(* IEC 61131-3 sources: AXOpen/src/components.festo.drives/ctrl/src/AxoCmmtAs (part 7) *)

            IF(_AxisReference = NULL) THEN
                RETURN;
            END_IF;

            IF Enable THEN
                Busy := TRUE;
                IF VelocityFactor <= 0.0 OR  VelocityFactor >= 2.0 OR AccelerationFactor <= 0.0 OR  AccelerationFactor > 1.0 OR JerkFactor <= 0.0 OR  JerkFactor > 1.0 THEN
                    Error := TRUE;
                ELSE
                    _AxisReference^.Data.OverrideVelocityFactor := VelocityFactor;
                    _AxisReference^.Data.OverrideAccelerationFactor := AccelerationFactor;
                    _AxisReference^.Data.OverrideJerkFactor := JerkFactor;
                    _AxisReference^.Telegram111_Out.Override_ := TO_WORD(TO_INT(16384.0/VelocityFactor));
                    Enabled	:= TRUE;
                END_IF;
            END_IF;
        END_METHOD

        ///<summary>
        /// This method returns the value of a vendor specific parameter. The returned Value has to be converted to Real
        /// if necessary. If not possible, the vendor has to supply a vendor specific method to read the parameter.
        ///<summary>
        VAR INTERNAL
            MC_ReadParameterEnable_PV       : 	BOOL := FALSE;		//Enable - previous value
            MC_ReadParameterErrorID         : 	WORD;
            MC_ReadParameterCycle			: 	ULINT;
            MC_ReadParameterValue			: 	LINT;
            MC_ReadParameterValid			: 	BOOL;
        END_VAR
        METHOD PUBLIC OVERRIDE MC_ReadParameter
            VAR_INPUT
                AxisRef         :   AXOpen.Components.Abstractions.Drives.IAxoAxisReference;
                Enable          :   BOOL;                       //  Get the value of the parameter continuously while enabled
                ParameterNumber :   DINT;                       //  Number of the parameter. One can also use symbolic parameter names which are declared as VAR CONST.
            END_VAR
            VAR_OUTPUT
                Valid           :   BOOL;                       //  A valid output is available at the method
                Busy            :   BOOL;                       //  The method is not finished and new output values are to be expected
                Error           :   BOOL;                       //  Signals that an error has occurred within the method
                ErrorID         :   WORD;                       //  Error identification
                Value           :   LINT;                       //  Value of the specified parameter in the datatype, as specified by the vendor
            END_VAR
            VAR
                _AxisReference :  REF_TO AXOpen.Components.Festo.Drives.AxoCmmtAsAxisReference;
                Dummy : BOOL;
            END_VAR

            _AxisReference ?= AxisRef;

            Messenger.ActivateOnCondition(ULINT#720,_AxisReference = NULL, eAxoMessageCategory#ProgrammingError);

            IF(_AxisReference = NULL) THEN
                RETURN;
            END_IF;

            IF Enable AND NOT MC_ReadParameterEnable_PV AND State = UINT#0 THEN
                _AxisReference^.Status.CurrentMotionTaskId := AXOpen.Components.Drives.eAxoMotionTaskId#Axo_ReadParameter;
                _AxisReference^.Data.Cycle := _AxisReference^.Data.Cycle + ULINT#2;
                MC_ReadParameterCycle := _AxisReference^.Data.Cycle ;
            END_IF;

            IF Enable THEN
                IF State = UINT#0 THEN
                    Busy := TRUE;
                    MC_ReadParameterErrorID := WORD#16#0000;
                    Parametrization.Inputs.Enable := FALSE;
                    State := UINT#160;
                END_IF;
                IF State = UINT#160 THEN
                    Busy := TRUE;
                    Parametrization.Inputs.Enable := TRUE;
                    Parametrization.Inputs.ReadWrite   := FALSE;
                    Parametrization.Inputs.ParameterNo := TO_INT(ParameterNumber);
                    Parametrization.Inputs.Subindex    := 0;
                    Parametrization.Inputs.AxisNo  := BYTE#1;
                    Parametrization.Inputs.HardwareId  := _AxisReference^.Data.MAP_HW_ID;
                    IF Parametrization.Outputs.Done AND NOT Parametrization.Outputs.Error THEN
                        MC_ReadParameterValid := TRUE;
                        MC_ReadParameterValue := Parametrization.Outputs.ValueReadLINT;
                        State := UINT#161;
                    END_IF;
                    IF Parametrization.Outputs.Error THEN
                        MC_MoveVelocityErrorID := WORD#801;
                        State := UINT#169;
                    END_IF;
                END_IF;
                IF State = UINT#161 THEN
                    Busy := TRUE;
                    Parametrization.Inputs.Enable := FALSE;
                    Parametrization.Inputs.ReadWrite   := FALSE;
                    IF  NOT Parametrization.Outputs.Done THEN
                        State := UINT#160;
                    END_IF;
                END_IF;
                IF State = UINT#169 THEN
                    Error := TRUE;
                END_IF;

                IF State>=UINT#160 AND State<UINT#167 THEN
                    IF _AxisReference^.Data.Cycle <> MC_ReadParameterCycle THEN
                        _AxisReference^.Data.Cycle := _AxisReference^.Data.Cycle - ULINT#1;
                        State := UINT#169;
                    END_IF;
                END_IF;
            END_IF;

            IF NOT Enable AND MC_ReadParameterEnable_PV  THEN
                _AxisReference^.Status.CurrentMotionTaskId := AXOpen.Components.Drives.eAxoMotionTaskId#Axo_None;
                MC_ReadParameterErrorID := WORD#0;
                MC_ReadParameterCycle := ULINT#0;
                MC_ReadParameterValid := FALSE;
                MC_ReadParameterValue := LINT#0;
                State := UINT#0;
            END_IF;

            ErrorID := MC_ReadParameterErrorID;
            Valid := MC_ReadParameterValid;
            Value := MC_ReadParameterValue;
            MC_ReadParameterEnable_PV := Enable;
        END_METHOD

        ///<summary>
        /// This method returns the value of a vendor specific parameter with datatype REAL.
        ///<summary>
        VAR INTERNAL
            MC_ReadRealParameterEnable_PV       : 	BOOL := FALSE;		//Enable - previous value
            MC_ReadRealParameterErrorID         : 	WORD;
            MC_ReadRealParameterCycle			: 	ULINT;
            MC_ReadRealParameterValue			: 	REAL;
            MC_ReadRealParameterValid			: 	BOOL;
        END_VAR
        METHOD PUBLIC OVERRIDE MC_ReadRealParameter
            VAR_INPUT
                AxisRef         :   AXOpen.Components.Abstractions.Drives.IAxoAxisReference;
                Enable          :   BOOL;                       //  Get the value of the parameter continuously while enabled
                ParameterNumber :   DINT;                       //  Number of the parameter. One can also use symbolic parameter names which are declared as VAR CONST.
            END_VAR
            VAR_OUTPUT
                Valid           :   BOOL;                       //  A valid output is available at the method
                Busy            :   BOOL;                       //  The method is not finished and new output values are to be expected
                Error           :   BOOL;                       //  Signals that an error has occurred within the method
                ErrorID         :   WORD;                       //  Error identification
                Value           :   REAL;                       //  Value of the specified parameter in the datatype, as specified by the vendor
            END_VAR
            VAR
                _AxisReference :  REF_TO AXOpen.Components.Festo.Drives.AxoCmmtAsAxisReference;
                Dummy : BOOL;
            END_VAR

            _AxisReference ?= AxisRef;

            Messenger.ActivateOnCondition(ULINT#721,_AxisReference = NULL, eAxoMessageCategory#ProgrammingError);

            IF(_AxisReference = NULL) THEN
                RETURN;
            END_IF;
            IF Enable AND NOT MC_ReadRealParameterEnable_PV AND State = UINT#0 THEN
                _AxisReference^.Status.CurrentMotionTaskId := AXOpen.Components.Drives.eAxoMotionTaskId#Axo_ReadRealParameter;
                _AxisReference^.Data.Cycle := _AxisReference^.Data.Cycle + ULINT#2;
                MC_ReadRealParameterCycle := _AxisReference^.Data.Cycle ;
            END_IF;

            IF Enable THEN
                IF State = UINT#0 THEN
                    Busy := TRUE;
                    MC_ReadRealParameterErrorID := WORD#16#0000;
                    Parametrization.Inputs.Enable := FALSE;
                    State := UINT#170;
                END_IF;
                IF State = UINT#170 THEN
                    Busy := TRUE;
                    Parametrization.Inputs.Enable := TRUE;
                    Parametrization.Inputs.ReadWrite   := FALSE;
                    Parametrization.Inputs.ParameterNo := TO_INT(ParameterNumber);
                    Parametrization.Inputs.Subindex    := 0;
                    Parametrization.Inputs.AxisNo  := BYTE#1;
                    Parametrization.Inputs.HardwareId  := _AxisReference^.Data.MAP_HW_ID;
                    IF Parametrization.Outputs.Done AND NOT Parametrization.Outputs.Error THEN
                        MC_ReadRealParameterValid := TRUE;
                        MC_ReadRealParameterValue := Parametrization.Outputs.ValueReadREAL;
                        State := UINT#171;
                    END_IF;
                    IF Parametrization.Outputs.Error THEN
                        MC_MoveVelocityErrorID := WORD#802;
                        State := UINT#179;
                    END_IF;
                END_IF;
                IF State = UINT#171 THEN
                    Busy := TRUE;
                    Parametrization.Inputs.Enable := FALSE;
                    Parametrization.Inputs.ReadWrite   := FALSE;
                    IF  NOT Parametrization.Outputs.Done THEN
                        State := UINT#170;
                    END_IF;
                END_IF;
                IF State = UINT#179 THEN
                    Error := TRUE;
                END_IF;

                IF State>=UINT#170 AND State<UINT#177 THEN
                    IF _AxisReference^.Data.Cycle <> MC_ReadRealParameterCycle THEN
                        _AxisReference^.Data.Cycle := _AxisReference^.Data.Cycle - ULINT#1;
                        State := UINT#179;
                    END_IF;
                END_IF;
            END_IF;

            IF NOT Enable AND MC_ReadRealParameterEnable_PV  THEN
                _AxisReference^.Status.CurrentMotionTaskId := AXOpen.Components.Drives.eAxoMotionTaskId#Axo_None;
                MC_ReadRealParameterErrorID := WORD#0;
                MC_ReadRealParameterCycle := ULINT#0;
                MC_ReadRealParameterValid := FALSE;
                MC_ReadRealParameterValue := REAL#0.0;
                State := UINT#0;
            END_IF;

            ErrorID := MC_ReadRealParameterErrorID;
            Valid := MC_ReadRealParameterValid;
            Value := MC_ReadRealParameterValue;
            MC_ReadRealParameterEnable_PV := Enable;
        END_METHOD

        ///<summary>
        /// This method returns the value of a vendor specific parameter with datatype BOOL.
        ///<summary>
        VAR INTERNAL
            MC_ReadBoolParameterEnable_PV       : 	BOOL := FALSE;		//Enable - previous value
            MC_ReadBoolParameterErrorID         : 	WORD;
            MC_ReadBoolParameterCycle			: 	ULINT;
            MC_ReadBoolParameterValue			: 	BOOL;
            MC_ReadBoolParameterValid			: 	BOOL;
        END_VAR
        METHOD PUBLIC OVERRIDE MC_ReadBoolParameter
            VAR_INPUT
                AxisRef         :   AXOpen.Components.Abstractions.Drives.IAxoAxisReference;
                Enable          :   BOOL;                       //  Get the value of the parameter continuously while enabled
                ParameterNumber :   DINT;                       //  Number of the parameter. One can also use symbolic parameter names which are declared as VAR CONST.
            END_VAR
            VAR_OUTPUT
                Valid           :   BOOL;                       //  A valid output is available at the method
                Busy            :   BOOL;                       //  The method is not finished and new output values are to be expected
                Error           :   BOOL;                       //  Signals that an error has occurred within the method
                ErrorID         :   WORD;                       //  Error identification
                Value           :   BOOL;                       //  Value of the specified parameter in the datatype, as specified by the vendor
            END_VAR
            VAR
                _AxisReference :  REF_TO AXOpen.Components.Festo.Drives.AxoCmmtAsAxisReference;
                Dummy : BOOL;
            END_VAR
            RETURN;

            _AxisReference ?= AxisRef;

            Messenger.ActivateOnCondition(ULINT#722,_AxisReference = NULL, eAxoMessageCategory#ProgrammingError);

            IF(_AxisReference = NULL) THEN
                RETURN;
            END_IF;

            IF Enable AND NOT MC_ReadBoolParameterEnable_PV AND State = UINT#0 THEN
                _AxisReference^.Status.CurrentMotionTaskId := AXOpen.Components.Drives.eAxoMotionTaskId#Axo_ReadBoolParameter;
                _AxisReference^.Data.Cycle := _AxisReference^.Data.Cycle + ULINT#2;
                MC_ReadBoolParameterCycle := _AxisReference^.Data.Cycle ;
            END_IF;

            IF Enable THEN
                IF State = UINT#0 THEN
                    Busy := TRUE;
                    MC_ReadBoolParameterErrorID := WORD#16#0000;
                    Parametrization.Inputs.Enable := FALSE;
                    State := UINT#180;
                END_IF;
                IF State = UINT#180 THEN
                    Busy := TRUE;
                    Parametrization.Inputs.Enable := TRUE;
                    Parametrization.Inputs.ReadWrite   := FALSE;
                    Parametrization.Inputs.ParameterNo := TO_INT(ParameterNumber);
                    Parametrization.Inputs.Subindex    := 0;
                    Parametrization.Inputs.AxisNo  := BYTE#1;
                    Parametrization.Inputs.HardwareId  := _AxisReference^.Data.MAP_HW_ID;
                    IF Parametrization.Outputs.Done AND NOT Parametrization.Outputs.Error THEN
                        MC_ReadBoolParameterValid := TRUE;
                        MC_ReadBoolParameterValue := Parametrization.Outputs.ValueReadBOOL;
                        State := UINT#181;
                    END_IF;
                    IF Parametrization.Outputs.Error THEN
                        MC_MoveVelocityErrorID := WORD#801;
                        State := UINT#189;
                    END_IF;
                END_IF;
                IF State = UINT#181 THEN
                    Busy := TRUE;
                    Parametrization.Inputs.Enable := FALSE;
                    Parametrization.Inputs.ReadWrite   := FALSE;
                    IF  NOT Parametrization.Outputs.Done THEN
                        State := UINT#180;
                    END_IF;
                END_IF;
                IF State = UINT#189 THEN
                    Error := TRUE;
                END_IF;

                IF State>=UINT#180 AND State<UINT#187 THEN
                    IF _AxisReference^.Data.Cycle <> MC_ReadBoolParameterCycle THEN
                        _AxisReference^.Data.Cycle := _AxisReference^.Data.Cycle - ULINT#1;
                        State := UINT#189;
                    END_IF;
                END_IF;
            END_IF;

            IF NOT Enable AND MC_ReadBoolParameterEnable_PV  THEN
                _AxisReference^.Status.CurrentMotionTaskId := AXOpen.Components.Drives.eAxoMotionTaskId#Axo_None;
                MC_ReadBoolParameterErrorID := WORD#0;
                MC_ReadBoolParameterCycle := ULINT#0;
                MC_ReadBoolParameterValid := FALSE;
                MC_ReadBoolParameterValue := FALSE;
                State := UINT#0;
            END_IF;

            ErrorID := MC_ReadBoolParameterErrorID;
            Valid := MC_ReadBoolParameterValid;
            Value := MC_ReadBoolParameterValue;
            MC_ReadBoolParameterEnable_PV := Enable;

        END_METHOD

        ///<summary>
        /// This method modifies the value of a vendor specific parameter.
        ///<summary>
        VAR INTERNAL
            MC_WriteParameterExecute_PV     : 	BOOL := FALSE;		//Enable - previous value
            MC_WriteParameterErrorID        : 	WORD;
            MC_WriteParameterCycle			: 	ULINT;
        END_VAR
        METHOD PUBLIC OVERRIDE MC_WriteParameter
            VAR_INPUT
                AxisRef         :   AXOpen.Components.Abstractions.Drives.IAxoAxisReference;
                Execute         :   BOOL;                       //  Write the value of the parameter at rising edge
                ParameterNumber :   DINT;                       //  Number of the parameter (correspondence between number andparameter is specified in the table above)
                Value           :   LINT;                       //  New value of the specified parameter
                ExecutionMode   :   AXOpen.Components.Abstractions.Drives.eAxoExecutionMode;          //  Defines the chronological sequence of the method.
            END_VAR
            VAR_OUTPUT
                Done            :   BOOL;                       //  Parameter successfully written
                Busy            :   BOOL;                       //  The method is not finished and new output values are to be expected.
                Error           :   BOOL;                       //  Signals that an error has occurred within the method
                ErrorID         :   WORD;                       //  Error identification
            END_VAR
            VAR
                _AxisReference :  REF_TO AXOpen.Components.Festo.Drives.AxoCmmtAsAxisReference;
                Dummy : BOOL;
            END_VAR

            _AxisReference ?= AxisRef;

            Messenger.ActivateOnCondition(ULINT#723,_AxisReference = NULL, eAxoMessageCategory#ProgrammingError);

            IF(_AxisReference = NULL) THEN
                RETURN;
            END_IF;

            IF THIS.AxoWriteParameter_Task.StartTriggered()  THEN
                _AxisReference^.Status.CurrentMotionTaskId := AXOpen.Components.Drives.eAxoMotionTaskId#Axo_WriteParameter;
            END_IF;

            IF Execute AND NOT MC_WriteParameterExecute_PV AND State = UINT#0 THEN
                _AxisReference^.Data.Cycle := _AxisReference^.Data.Cycle + ULINT#2;
                MC_WriteParameterCycle := _AxisReference^.Data.Cycle ;
            END_IF;

            IF Execute THEN
                IF State = UINT#0 THEN
                    Busy := TRUE;
                    Parametrization.Inputs.Enable := FALSE;
                    State := UINT#190;
                END_IF;
                IF State = UINT#190 THEN
                    Busy := TRUE;
                    Parametrization.Inputs.Enable := TRUE;
                    Parametrization.Inputs.ReadWrite   := TRUE;
                    Parametrization.Inputs.ParameterNo := TO_INT(ParameterNumber);
                    Parametrization.Inputs.Subindex    := 0;
                    Parametrization.Inputs.AxisNo  := BYTE#1;
                    Parametrization.Inputs.HardwareId  := _AxisReference^.Data.MAP_HW_ID;
                    Parametrization.Inputs.ValueWriteLINT := Value;
                    IF Parametrization.Outputs.Done AND NOT Parametrization.Outputs.Error THEN
                        State := UINT#191;
                    END_IF;
                    IF Parametrization.Outputs.Error THEN
                        MC_WriteParameterErrorID := WORD#804;
                        State := UINT#199;
                    END_IF;
                END_IF;
                IF State = UINT#191 THEN
                    Busy := TRUE;
                    Parametrization.Inputs.Enable := FALSE;
                    Parametrization.Inputs.ReadWrite   := FALSE;
                    IF  NOT Parametrization.Outputs.Done THEN
                        State := UINT#197;
                    END_IF;
                END_IF;
                IF State = UINT#197 THEN
                    Done := TRUE;
                    MC_WriteParameterCycle := ULINT#0;
                END_IF;
                IF State = UINT#199 THEN
                    MC_WriteParameterCycle := ULINT#0;
                    Error := TRUE;
                END_IF;

                IF State>=UINT#190 AND State<UINT#197 THEN
                    IF _AxisReference^.Data.Cycle <> MC_WriteParameterCycle THEN
                        _AxisReference^.Data.Cycle := _AxisReference^.Data.Cycle - ULINT#1;
                        State := UINT#199;
                    END_IF;
                END_IF;
            END_IF;

            IF THIS.AxoWriteParameter_Task.DoneReached() THEN
                _AxisReference^.Status.CurrentMotionTaskId := AXOpen.Components.Drives.eAxoMotionTaskId#Axo_Done;
                MC_WriteParameterErrorID := WORD#0;
                // MC_WriteParameterCycle := ULINT#0;
                State := UINT#0;
            END_IF;

            IF THIS.AxoWriteParameter_Task.RestoreTriggered() AND State>=UINT#190 AND State<=UINT#199 THEN
                _AxisReference^.Status.CurrentMotionTaskId := AXOpen.Components.Drives.eAxoMotionTaskId#Axo_None;
                MC_WriteParameterErrorID := WORD#0;
                MC_WriteParameterCycle := ULINT#0;
                State := UINT#0;
            END_IF;

            ErrorID := MC_WriteParameterErrorID;
            MC_WriteParameterExecute_PV := Execute;
        END_METHOD

        ///<summary>
        /// This method modifies the value of a vendor specific parameter of type Real.
        ///<summary>
        VAR INTERNAL
            MC_WriteRealParameterExecute_PV     : 	BOOL := FALSE;		//Enable - previous value
            MC_WriteRealParameterErrorID        : 	WORD;
            MC_WriteRealParameterCycle			: 	ULINT;
        END_VAR
        METHOD PUBLIC OVERRIDE MC_WriteRealParameter
            VAR_INPUT
                AxisRef         :   AXOpen.Components.Abstractions.Drives.IAxoAxisReference;
                Execute         :   BOOL;                       //  Write the value of the parameter at rising edge
                ParameterNumber :   DINT;                       //  Number of the parameter (correspondence between number andparameter is specified in the table above)
                Value           :   REAL;                       //  New value of the specified parameter
                ExecutionMode   :   AXOpen.Components.Abstractions.Drives.eAxoExecutionMode;          //  Defines the chronological sequence of the method.
            END_VAR
            VAR_OUTPUT
                Done            :   BOOL;                       //  Parameter successfully written
                Busy            :   BOOL;                       //  The method is not finished and new output values are to be expected.
                Error           :   BOOL;                       //  Signals that an error has occurred within the method
                ErrorID         :   WORD;                       //  Error identification
            END_VAR
            VAR
                _AxisReference :  REF_TO AXOpen.Components.Festo.Drives.AxoCmmtAsAxisReference;
                Dummy : BOOL;
            END_VAR

            _AxisReference ?= AxisRef;

            Messenger.ActivateOnCondition(ULINT#724,_AxisReference = NULL, eAxoMessageCategory#ProgrammingError);

            IF(_AxisReference = NULL) THEN
                RETURN;
            END_IF;

            IF THIS.AxoWriteRealParameter_Task.StartTriggered()  THEN
                _AxisReference^.Status.CurrentMotionTaskId := AXOpen.Components.Drives.eAxoMotionTaskId#Axo_WriteRealParameter;
            END_IF;

            IF Execute AND NOT MC_WriteRealParameterExecute_PV AND State = UINT#0 THEN
                _AxisReference^.Data.Cycle := _AxisReference^.Data.Cycle + ULINT#2;
                MC_WriteRealParameterCycle := _AxisReference^.Data.Cycle ;
            END_IF;

            IF Execute THEN
                IF State = UINT#0 THEN
                    Busy := TRUE;
                    Parametrization.Inputs.Enable := FALSE;
                    State := UINT#200;
                END_IF;
                IF State = UINT#200 THEN
                    Busy := TRUE;
                    Parametrization.Inputs.Enable := TRUE;
                    Parametrization.Inputs.ReadWrite   := TRUE;
                    Parametrization.Inputs.ParameterNo := TO_INT(ParameterNumber);
                    Parametrization.Inputs.Subindex    := 0;
                    Parametrization.Inputs.AxisNo  := BYTE#1;
                    Parametrization.Inputs.HardwareId  := _AxisReference^.Data.MAP_HW_ID;
                    Parametrization.Inputs.ValueWriteREAL := Value;
                    IF Parametrization.Outputs.Done AND NOT Parametrization.Outputs.Error THEN
                        State := UINT#201;
                    END_IF;
                    IF Parametrization.Outputs.Error THEN
                        MC_WriteRealParameterErrorID := WORD#805;
                        State := UINT#209;
                    END_IF;
                END_IF;
                IF State = UINT#201 THEN
                    Busy := TRUE;
                    Parametrization.Inputs.Enable := FALSE;
                    Parametrization.Inputs.ReadWrite   := FALSE;
                    IF  NOT Parametrization.Outputs.Done THEN
                        State := UINT#207;
                    END_IF;
                END_IF;
                IF State = UINT#207 THEN
                    Done := TRUE;
                    MC_WriteRealParameterCycle := ULINT#0;
                END_IF;
                IF State = UINT#209 THEN
                    MC_WriteRealParameterCycle := ULINT#0;
                    Error := TRUE;
                END_IF;

                IF State>=UINT#200 AND State<UINT#207 THEN
                    IF _AxisReference^.Data.Cycle <> MC_WriteRealParameterCycle THEN
                        _AxisReference^.Data.Cycle := _AxisReference^.Data.Cycle - ULINT#1;
                        State := UINT#209;
                    END_IF;
                END_IF;
            END_IF;

            IF THIS.AxoWriteRealParameter_Task.DoneReached() THEN
                _AxisReference^.Status.CurrentMotionTaskId := AXOpen.Components.Drives.eAxoMotionTaskId#Axo_Done;
                MC_WriteRealParameterErrorID := WORD#0;
                // MC_WriteRealParameterCycle := ULINT#0;
                State := UINT#0;
            END_IF;

            IF THIS.AxoWriteRealParameter_Task.RestoreTriggered() AND State>=UINT#200 AND State<=UINT#209 THEN
                _AxisReference^.Status.CurrentMotionTaskId := AXOpen.Components.Drives.eAxoMotionTaskId#Axo_None;
                MC_WriteRealParameterErrorID := WORD#0;
                MC_WriteRealParameterCycle := ULINT#0;
                State := UINT#0;
            END_IF;

            ErrorID := MC_WriteRealParameterErrorID;
            MC_WriteRealParameterExecute_PV := Execute;
        END_METHOD

        ///<summary>
        /// This method modifies the value of a vendor specific parameter of type BOOL.
        ///<summary>
        VAR INTERNAL
            MC_WriteBoolParameterExecute_PV     : 	BOOL := FALSE;		//Enable - previous value
            MC_WriteBoolParameterErrorID        : 	WORD;
            MC_WriteBoolParameterCycle			: 	ULINT;
        END_VAR
        METHOD PUBLIC OVERRIDE MC_WriteBoolParameter
            VAR_INPUT
                AxisRef         :   AXOpen.Components.Abstractions.Drives.IAxoAxisReference;
                Execute         :   BOOL;                       //  Write the value of the parameter at rising edge
                ParameterNumber :   DINT;                       //  Number of the parameter (correspondence between number andparameter is specified in the table above)
                Value           :   BOOL;                       //  New value of the specified parameter
                ExecutionMode   :   AXOpen.Components.Abstractions.Drives.eAxoExecutionMode;          //  Defines the chronological sequence of the method.
            END_VAR
            VAR_OUTPUT
                Done            :   BOOL;                       //  Parameter successfully written
                Busy            :   BOOL;                       //  The method is not finished and new output values are to be expected.
                Error           :   BOOL;                       //  Signals that an error has occurred within the method
                ErrorID         :   WORD;                       //  Error identification
            END_VAR
            VAR
                _AxisReference :  REF_TO AXOpen.Components.Festo.Drives.AxoCmmtAsAxisReference;
                Dummy : BOOL;
            END_VAR

            _AxisReference ?= AxisRef;

            Messenger.ActivateOnCondition(ULINT#725,_AxisReference = NULL, eAxoMessageCategory#ProgrammingError);

            IF(_AxisReference = NULL) THEN
                RETURN;
            END_IF;

            IF THIS.AxoWriteBoolParameter_Task.StartTriggered()  THEN
                _AxisReference^.Status.CurrentMotionTaskId := AXOpen.Components.Drives.eAxoMotionTaskId#Axo_WriteBoolParameter;
            END_IF;

            IF Execute AND NOT MC_WriteBoolParameterExecute_PV AND State = UINT#0 THEN
                _AxisReference^.Data.Cycle := _AxisReference^.Data.Cycle + ULINT#2;
                MC_WriteBoolParameterCycle := _AxisReference^.Data.Cycle ;
            END_IF;

            IF Execute THEN
                IF State = UINT#0 THEN
                    Busy := TRUE;
                    Parametrization.Inputs.Enable := FALSE;
                    State := UINT#210;
                END_IF;
                IF State = UINT#210 THEN
                    Busy := TRUE;
                    Parametrization.Inputs.Enable := TRUE;
                    Parametrization.Inputs.ReadWrite   := TRUE;
                    Parametrization.Inputs.ParameterNo := TO_INT(ParameterNumber);
                    Parametrization.Inputs.Subindex    := 0;
                    Parametrization.Inputs.AxisNo  := BYTE#1;
                    Parametrization.Inputs.HardwareId  := _AxisReference^.Data.MAP_HW_ID;
                    Parametrization.Inputs.ValueWriteBOOL := Value;
                    IF Parametrization.Outputs.Done AND NOT Parametrization.Outputs.Error THEN
                        State := UINT#211;
                    END_IF;
                    IF Parametrization.Outputs.Error THEN
                        MC_WriteBoolParameterErrorID := WORD#805;
                        State := UINT#219;
                    END_IF;
                END_IF;
                IF State = UINT#211 THEN
                    Busy := TRUE;
                    Parametrization.Inputs.Enable := FALSE;
                    Parametrization.Inputs.ReadWrite   := FALSE;
                    IF  NOT Parametrization.Outputs.Done THEN
                        State := UINT#217;
                    END_IF;
                END_IF;
                IF State = UINT#217 THEN
                    Done := TRUE;
                    MC_WriteBoolParameterCycle := ULINT#0;
                END_IF;
                IF State = UINT#219 THEN
                    MC_WriteBoolParameterCycle := ULINT#0;
                    Error := TRUE;
                END_IF;

                IF State>=UINT#210 AND State<UINT#217 THEN
                    IF _AxisReference^.Data.Cycle <> MC_WriteBoolParameterCycle THEN
                        _AxisReference^.Data.Cycle := _AxisReference^.Data.Cycle - ULINT#1;
                        State := UINT#219;
                    END_IF;
                END_IF;
            END_IF;

            IF THIS.AxoWriteBoolParameter_Task.DoneReached() THEN
                _AxisReference^.Status.CurrentMotionTaskId := AXOpen.Components.Drives.eAxoMotionTaskId#Axo_Done;
                MC_WriteBoolParameterErrorID := WORD#0;
                // MC_WriteBoolParameterCycle := ULINT#0;
                State := UINT#0;
            END_IF;

            IF THIS.AxoWriteBoolParameter_Task.RestoreTriggered() AND State>=UINT#210 AND State<=UINT#219 THEN
                _AxisReference^.Status.CurrentMotionTaskId := AXOpen.Components.Drives.eAxoMotionTaskId#Axo_None;
                MC_WriteBoolParameterErrorID := WORD#0;
                MC_WriteBoolParameterCycle := ULINT#0;
                State := UINT#0;
            END_IF;

            ErrorID := MC_WriteBoolParameterErrorID;
            MC_WriteBoolParameterExecute_PV := Execute;
        END_METHOD

        ///<summary>
        /// This method gives access to the value of the input, referenced by the datatype MC_INPUT_REF.
        /// It provides the value of the referenced input (BOOL).
        ///<summary>
        VAR INTERNAL
            MC_ReadDigitalInputEnable_PV        : 	BOOL := FALSE;		//Enable - previous value
            MC_ReadDigitalInputErrorID          : 	WORD;
            MC_ReadDigitalInputCycle			: 	ULINT;
            MC_ReadDigitalInputValue			: 	BOOL;
            MC_ReadDigitalInputValid			: 	BOOL;
        END_VAR
        METHOD PUBLIC OVERRIDE MC_ReadDigitalInput
            VAR_INPUT
                AxisRef         :   AXOpen.Components.Abstractions.Drives.IAxoAxisReference;
                Enable          :   BOOL;                       //  Get the value of the selected input signal continuously while enabled
                InputNumber     :   INT;                        //  Selects the input. Can be part of MC_INPUT_REF, if only one single input is referenced.
            END_VAR
            VAR_OUTPUT
                Valid           :   BOOL;                       //  A valid output is available at the method
                Busy            :   BOOL;                       //  The method is not finished and new output values are to be expected
                Error           :   BOOL;                       //  Signals that an error has occurred within the method
                ErrorID         :   WORD;                       //  Error identification
                Value           :   BOOL;                       //  The value of the selected input signal
            END_VAR
            VAR
                _AxisReference :  REF_TO AXOpen.Components.Festo.Drives.AxoCmmtAsAxisReference;
                Dummy : BOOL;
            END_VAR

            _AxisReference ?= AxisRef;

            Messenger.ActivateOnCondition(ULINT#726,_AxisReference = NULL, eAxoMessageCategory#ProgrammingError);

            IF(_AxisReference = NULL) THEN
                RETURN;
            END_IF;

            IF Enable AND NOT MC_ReadDigitalInputEnable_PV AND State = UINT#0 THEN
                _AxisReference^.Status.CurrentMotionTaskId := AXOpen.Components.Drives.eAxoMotionTaskId#Axo_ReadDigitalInput;
                _AxisReference^.Data.Cycle := _AxisReference^.Data.Cycle + ULINT#2;
                MC_ReadDigitalInputCycle := _AxisReference^.Data.Cycle ;
            END_IF;

            IF Enable THEN
                IF State = UINT#0 THEN
                    Busy := TRUE;
                    MC_ReadDigitalInputErrorID := WORD#16#0000;
                    Parametrization.Inputs.Enable := FALSE;
                    State := UINT#220;
                END_IF;
                IF State = UINT#220 THEN
                    Busy := TRUE;
                    Parametrization.Inputs.Enable := TRUE;
                    Parametrization.Inputs.ReadWrite   := FALSE;
                    Parametrization.Inputs.ParameterNo := 2888;
                    Parametrization.Inputs.Subindex    := 0;
                    Parametrization.Inputs.AxisNo  := BYTE#1;
                    Parametrization.Inputs.HardwareId  := _AxisReference^.Data.MAP_HW_ID;
                    IF Parametrization.Outputs.Done AND NOT Parametrization.Outputs.Error THEN
                        MC_ReadDigitalInputValid := TRUE;
                        MC_ReadDigitalInputValue := GetBit(TO_LWORD(Parametrization.Outputs.ValueReadLINT), TO_USINT(InputNumber));
                        State := UINT#221;
                    END_IF;
                    IF Parametrization.Outputs.Error THEN
                        MC_MoveVelocityErrorID := WORD#807;
                        State := UINT#229;
                    END_IF;
                END_IF;
                IF State = UINT#221 THEN
                    Busy := TRUE;
                    Parametrization.Inputs.Enable := FALSE;
                    Parametrization.Inputs.ReadWrite   := FALSE;
                    IF  NOT Parametrization.Outputs.Done THEN
                        State := UINT#220;
                    END_IF;
                END_IF;
                IF State = UINT#229 THEN
                    Error := TRUE;
                END_IF;

                IF State>=UINT#220 AND State<UINT#227 THEN
                    IF _AxisReference^.Data.Cycle <> MC_ReadDigitalInputCycle THEN
                        _AxisReference^.Data.Cycle := _AxisReference^.Data.Cycle - ULINT#1;
                        State := UINT#229;
                    END_IF;
                END_IF;
            END_IF;

            IF NOT Enable AND MC_ReadDigitalInputEnable_PV  THEN
                _AxisReference^.Status.CurrentMotionTaskId := AXOpen.Components.Drives.eAxoMotionTaskId#Axo_None;
                MC_ReadDigitalInputErrorID := WORD#0;
                MC_ReadDigitalInputCycle := ULINT#0;
                MC_ReadDigitalInputValid := FALSE;
                MC_ReadDigitalInputValue := FALSE;
                State := UINT#0;
            END_IF;

            ErrorID := MC_ReadDigitalInputErrorID;
            Valid := MC_ReadDigitalInputValid;
            Value := MC_ReadDigitalInputValue;
            MC_ReadDigitalInputEnable_PV := Enable;
        END_METHOD

        ///<summary>
        /// This method provides access to the value of a digital output, referenced by the datatype MC_OUTPUT_REF.
        /// It provides the value of the referenced output (BOOL).
        ///<summary>
        VAR INTERNAL
            MC_ReadDigitalOutputEnable_PV        : 	BOOL := FALSE;		//Enable - previous value
            MC_ReadDigitalOutputErrorID          : 	WORD;
            MC_ReadDigitalOutputCycle			: 	ULINT;
            MC_ReadDigitalOutputValue			: 	BOOL;
            MC_ReadDigitalOutputValid			: 	BOOL;
        END_VAR
        METHOD PUBLIC OVERRIDE MC_ReadDigitalOutput
            VAR_INPUT
                AxisRef         :   AXOpen.Components.Abstractions.Drives.IAxoAxisReference;
                Enable          :   BOOL;                       //  Get the value of the selected output signal continuously while enabled
                OutputNumber    :   INT;                        //  Selects the output. Can be part of MC_OUTPUT_REF, if only one single output is referenced.
            END_VAR
            VAR_OUTPUT
                Valid           :   BOOL;                       //  A valid output is available at the method
                Busy            :   BOOL;                       //  The method is not finished and new output values are to be expected
                Error           :   BOOL;                       //  Signals that an error has occurred within the method
                ErrorID         :   WORD;                       //  Error identification
                Value           :   BOOL;                       //  The value of the selected output signal
            END_VAR
            VAR
                _AxisReference :  REF_TO AXOpen.Components.Festo.Drives.AxoCmmtAsAxisReference;
                Dummy : BOOL;
            END_VAR

            _AxisReference ?= AxisRef;

            Messenger.ActivateOnCondition(ULINT#727,_AxisReference = NULL, eAxoMessageCategory#ProgrammingError);

            IF(_AxisReference = NULL) THEN
                RETURN;
            END_IF;

            IF Enable AND NOT MC_ReadDigitalOutputEnable_PV AND State = UINT#0 THEN
                _AxisReference^.Status.CurrentMotionTaskId := AXOpen.Components.Drives.eAxoMotionTaskId#Axo_ReadDigitalOutput;
                _AxisReference^.Data.Cycle := _AxisReference^.Data.Cycle + ULINT#2;
                MC_ReadDigitalOutputCycle := _AxisReference^.Data.Cycle ;
            END_IF;

            IF Enable THEN
                IF State = UINT#0 THEN
                    Busy := TRUE;
                    MC_ReadDigitalOutputErrorID := WORD#16#0000;
                    Parametrization.Inputs.Enable := FALSE;
                    State := UINT#230;
                END_IF;
                IF State = UINT#230 THEN
                    Busy := TRUE;
                    Parametrization.Inputs.Enable := TRUE;
                    Parametrization.Inputs.ReadWrite   := FALSE;
                    Parametrization.Inputs.ParameterNo := 2888;
                    Parametrization.Inputs.Subindex    := 0;
                    Parametrization.Inputs.AxisNo  := BYTE#1;
                    Parametrization.Inputs.HardwareId  := _AxisReference^.Data.MAP_HW_ID;
                    IF Parametrization.Outputs.Done AND NOT Parametrization.Outputs.Error THEN
                        MC_ReadDigitalOutputValid := TRUE;
                        MC_ReadDigitalOutputValue := GetBit(TO_LWORD(Parametrization.Outputs.ValueReadLINT), TO_USINT(OutputNumber));
                        State := UINT#231;
                    END_IF;
                    IF Parametrization.Outputs.Error THEN
                        MC_MoveVelocityErrorID := WORD#809;
                        State := UINT#239;
                    END_IF;
                END_IF;
                IF State = UINT#231 THEN
                    Busy := TRUE;
                    Parametrization.Inputs.Enable := FALSE;
                    Parametrization.Inputs.ReadWrite   := FALSE;
                    IF  NOT Parametrization.Outputs.Done THEN
                        State := UINT#230;
                    END_IF;
                END_IF;
                IF State = UINT#239 THEN
                    Error := TRUE;
                END_IF;

                IF State>=UINT#230 AND State<UINT#237 THEN
                    IF _AxisReference^.Data.Cycle <> MC_ReadDigitalOutputCycle THEN
                        _AxisReference^.Data.Cycle := _AxisReference^.Data.Cycle - ULINT#1;
                        State := UINT#239;
                    END_IF;
                END_IF;
            END_IF;

            IF NOT Enable AND MC_ReadDigitalOutputEnable_PV  THEN
                _AxisReference^.Status.CurrentMotionTaskId := AXOpen.Components.Drives.eAxoMotionTaskId#Axo_None;
                MC_ReadDigitalOutputErrorID := WORD#0;
                MC_ReadDigitalOutputCycle := ULINT#0;
                MC_ReadDigitalOutputValid := FALSE;
                MC_ReadDigitalOutputValue := FALSE;
                State := UINT#0;
            END_IF;

            ErrorID := MC_ReadDigitalOutputErrorID;
            Valid := MC_ReadDigitalOutputValid;
            Value := MC_ReadDigitalOutputValue;
            MC_ReadDigitalOutputEnable_PV := Enable;
        END_METHOD

        ///<summary>
        /// This method writes a value to the output referenced by the argument ‘Output’ once (with rising edge of Execute)
        ///<summary>
        VAR INTERNAL
            MC_WriteDigitalOutputExecute_PV     : 	BOOL := FALSE;		//Enable - previous value
            MC_WriteDigitalOutputErrorID        : 	WORD;
            MC_WriteDigitalOutputCycle			: 	ULINT;
        END_VAR
        METHOD PUBLIC OVERRIDE MC_WriteDigitalOutput
            VAR_INPUT
                AxisRef         :   AXOpen.Components.Abstractions.Drives.IAxoAxisReference;
                Execute         :   BOOL;                       //  Write the value of the selected output
                OutputNumber    :   INT;                        //  Selects the output. Can be part of MC_OUTPUT_REF, if only one single output is referenced.
                Value           :   BOOL;                       //  The value of the selected output signal
                ExecutionMode   :   AXOpen.Components.Abstractions.Drives.eAxoExecutionMode;          //  Defines the chronological sequence of the method.
            END_VAR
            VAR_OUTPUT
                Done            :   BOOL;                       //  Writing of the output signal value is done
                Busy            :   BOOL;                       //  The method is not finished and new output values are to be expected.
                Error           :   BOOL;                       //  Signals that an error has occurred within the method
                ErrorID         :   WORD;                       //  Error identification
            END_VAR
            VAR
                _AxisReference :  REF_TO AXOpen.Components.Festo.Drives.AxoCmmtAsAxisReference;
                Dummy : BOOL;
                Valid_          :   BOOL;
                Error_          :   BOOL;
                ErrorID_        :   WORD;
            END_VAR

            _AxisReference ?= AxisRef;

            Messenger.ActivateOnCondition(ULINT#728,_AxisReference = NULL, eAxoMessageCategory#ProgrammingError);

            IF(_AxisReference = NULL) THEN
                RETURN;
            END_IF;

            IF THIS.AxoWriteDigitalOutput_Task.StartTriggered()  THEN
                _AxisReference^.Status.CurrentMotionTaskId := AXOpen.Components.Drives.eAxoMotionTaskId#Axo_WriteDigitalOutput;
            END_IF;

            IF Execute AND NOT MC_WriteDigitalOutputExecute_PV AND State = UINT#0 THEN
                _AxisReference^.Data.Cycle := _AxisReference^.Data.Cycle + ULINT#2;
                MC_WriteDigitalOutputCycle := _AxisReference^.Data.Cycle ;
            END_IF;

            IF Execute THEN
                IF State = UINT#0 THEN
                    Busy := TRUE;
                    Parametrization.Inputs.Enable := FALSE;
                    State := UINT#240;
                    //Remove after implementation on the drive side
                    State := UINT#249;
                    MC_WriteDigitalOutputErrorID := WORD#810;
                END_IF;
                IF State = UINT#240 THEN
                    Busy := TRUE;
                    Parametrization.Inputs.Enable := TRUE;
                    Parametrization.Inputs.ReadWrite   := TRUE;
                    Parametrization.Inputs.ParameterNo := 0;
                    Parametrization.Inputs.Subindex    := 0;
                    Parametrization.Inputs.AxisNo  := BYTE#1;
                    Parametrization.Inputs.HardwareId  := _AxisReference^.Data.MAP_HW_ID;
                    Parametrization.Inputs.ValueWriteBOOL := Value;
                    IF Parametrization.Outputs.Done AND NOT Parametrization.Outputs.Error THEN
                        State := UINT#241;
                    END_IF;
                    IF Parametrization.Outputs.Error THEN
                        MC_WriteDigitalOutputErrorID := WORD#811;
                        State := UINT#249;
                    END_IF;
                END_IF;
                IF State = UINT#241 THEN
                    Busy := TRUE;
                    Parametrization.Inputs.Enable := FALSE;
                    Parametrization.Inputs.ReadWrite   := FALSE;
                    IF  NOT Parametrization.Outputs.Done THEN
                        State := UINT#247;
                    END_IF;
                END_IF;
                IF State = UINT#247 THEN
                    Done := TRUE;
                    MC_WriteDigitalOutputCycle := ULINT#0;
                END_IF;
                IF State = UINT#249 THEN
                    MC_WriteDigitalOutputCycle := ULINT#0;
                    Error := TRUE;
                END_IF;

                IF State>=UINT#240 AND State<UINT#247 THEN
                    IF _AxisReference^.Data.Cycle <> MC_WriteDigitalOutputCycle THEN
                        _AxisReference^.Data.Cycle := _AxisReference^.Data.Cycle - ULINT#1;
                        State := UINT#249;
                    END_IF;
                END_IF;
            END_IF;

            IF THIS.AxoWriteDigitalOutput_Task.DoneReached() THEN
                _AxisReference^.Status.CurrentMotionTaskId := AXOpen.Components.Drives.eAxoMotionTaskId#Axo_Done;
                MC_WriteDigitalOutputErrorID := WORD#0;
                // MC_WriteDigitalOutputCycle := ULINT#0;
                State := UINT#0;
            END_IF;

            IF THIS.AxoWriteDigitalOutput_Task.RestoreTriggered() AND State>=UINT#240 AND State<=UINT#249 THEN
                _AxisReference^.Status.CurrentMotionTaskId := AXOpen.Components.Drives.eAxoMotionTaskId#Axo_None;
                MC_WriteDigitalOutputErrorID := WORD#0;
                MC_WriteDigitalOutputCycle := ULINT#0;
                State := UINT#0;
            END_IF;

            ErrorID := MC_WriteDigitalOutputErrorID;
            MC_WriteDigitalOutputExecute_PV := Execute;

        END_METHOD

        ///<summary>
        /// This method returns the actual position.
        ///<summary>
        METHOD PUBLIC OVERRIDE MC_ReadActualPosition
             VAR_INPUT
                AxisRef         :   AXOpen.Components.Abstractions.Drives.IAxoAxisReference;
                Enable          :   BOOL;                       //  Get the value of the parameter continuously while enabled
            END_VAR
            VAR_OUTPUT
                Valid           :   BOOL;                       //  A valid output is available at the method
                Busy            :   BOOL;                       //  The method is not finished and new output values are to be expected
                Error           :   BOOL;                       //  Signals that an error has occurred within the method
                ErrorID         :   WORD;                       //  Error identification
                Position        :   LREAL;                       //  New absolute position (in axis’ unit [u])
            END_VAR
            VAR
                _AxisReference :  REF_TO AXOpen.Components.Festo.Drives.AxoCmmtAsAxisReference;
                Dummy : BOOL;
            END_VAR

            _AxisReference ?= AxisRef;

            Messenger.ActivateOnCondition(ULINT#729,_AxisReference = NULL, eAxoMessageCategory#ProgrammingError);

            IF(_AxisReference = NULL) THEN
                RETURN;
            END_IF;

            IF Enable THEN
                Valid := TRUE;
                Position := THIS.ActualPosition;
            END_IF;
        END_METHOD

        ///<summary>
        /// This method returns the value of the actual velocity as long as ‘Enable’ is set. ‘Valid’ is true when the
        /// dataoutput ‘Velocity’ is valid. If ‘Enable’ is Reset, the data loses its validity, and all outputs are reset,
        /// no matter if new data is available.
        ///<summary>
        METHOD PUBLIC OVERRIDE MC_ReadActualVelocity
            VAR_INPUT
                AxisRef         :   AXOpen.Components.Abstractions.Drives.IAxoAxisReference;
                Enable          :   BOOL;                       //  Get the value of the parameter continuously while enabled
            END_VAR
            VAR_OUTPUT
                Valid           :   BOOL;                       //  A valid output is available at the method
                Busy            :   BOOL;                       //  The method is not finished and new output values are to be expected
                Error           :   BOOL;                       //  Signals that an error has occurred within the method
                ErrorID         :   WORD;                       //  Error identification
                Velocity        :   LREAL;                       //  The value of the actual velocity (in axis’ unit [u/s])
            END_VAR
            VAR
                _AxisReference :  REF_TO AXOpen.Components.Festo.Drives.AxoCmmtAsAxisReference;
                Dummy : BOOL;
            END_VAR

            _AxisReference ?= AxisRef;

            Messenger.ActivateOnCondition(ULINT#730,_AxisReference = NULL, eAxoMessageCategory#ProgrammingError);

            IF(_AxisReference = NULL) THEN
                RETURN;
            END_IF;

            IF Enable THEN
                Valid := TRUE;
                Velocity := THIS.ActualVelocity;
            END_IF;
        END_METHOD

        ///<summary>
        /// This method returns the value of the actual torque or force as long as ‘Enable’ is set. ‘Valid’ is true when the
        /// data-output ‘Torque’ is valid. If ‘Enable’ is Reset, the data loses its validity, and ‘Valid’ is also reset,
        /// no matter if new data is available.
        ///<summary>
        METHOD PUBLIC OVERRIDE MC_ReadActualTorque
            VAR_INPUT
                AxisRef         :   AXOpen.Components.Abstractions.Drives.IAxoAxisReference;
                Enable          :   BOOL;                       //  Get the value of the parameter continuously while enabled
            END_VAR
            VAR_OUTPUT
                Valid           :   BOOL;                       //  A valid output is available at the method
                Busy            :   BOOL;                       //  The method is not finished and new output values are to be expected
                Error           :   BOOL;                       //  Signals that an error has occurred within the method
                ErrorID         :   WORD;                       //  Error identification
                Torque          :   LREAL;                       //  The value of the actual torque or force (in technical units)
            END_VAR
            VAR
                _AxisReference :  REF_TO AXOpen.Components.Festo.Drives.AxoCmmtAsAxisReference;
                Dummy : BOOL;
            END_VAR

            _AxisReference ?= AxisRef;

            Messenger.ActivateOnCondition(ULINT#731,_AxisReference = NULL, eAxoMessageCategory#ProgrammingError);

            IF(_AxisReference = NULL) THEN
                RETURN;
            END_IF;
            IF Enable THEN
                Valid := TRUE;
                Torque := THIS.ActualTorque;
            END_IF;
        END_METHOD

        ///<summary>
        /// This method returns in detail the status of the state diagram of the axis
        ///<summary>
        VAR INTERNAL
            MC_ReadStatusEnable_PV				: 	BOOL := FALSE;		//Enable - previous value
            MC_ReadStatusDone_PV				:	BOOL := FALSE;		//Done - previous value
            MC_ReadStatusStateNumber			: 	INT; 				//Call number of the method MC_ReadRealParameter
        END_VAR
        METHOD PUBLIC OVERRIDE MC_ReadStatus
            VAR_INPUT
                AxisRef             :   AXOpen.Components.Abstractions.Drives.IAxoAxisReference;
                Enable              :   BOOL;                       //  Get the value of the parameter continuously while enabled
            END_VAR
            VAR_OUTPUT
                Valid               :   BOOL;                       //  A valid output is available at the method
                Busy                :   BOOL;                       //  The method is not finished and new output values are to be expected
                Error               :   BOOL;                       //  Signals that an error has occurred within the method
                ErrorID             :   WORD;                       //  Error identification
                ErrorStop           :   BOOL;                       //  See state diagram
                Disabled            :   BOOL;                       //  See state diagram
                Stopping            :   BOOL;                       //  See state diagram
                Homing              :   BOOL;                       //  See state diagram
                Standstill          :   BOOL;                       //  See state diagram
                DiscreteMotion      :   BOOL;                       //  See state diagram
                ContinuousMotion     :   BOOL;                       //  See state diagram
                SynchronizedMotion  : BOOL;                       //  See state diagram
            END_VAR
            VAR
                _AxisReference :  REF_TO AXOpen.Components.Festo.Drives.AxoCmmtAsAxisReference;
                Dummy : BOOL;
            END_VAR

            _AxisReference ?= AxisRef;

            Messenger.ActivateOnCondition(ULINT#732,_AxisReference = NULL, eAxoMessageCategory#ProgrammingError);

            IF(_AxisReference = NULL) THEN
                RETURN;
            END_IF;

            IF Enable THEN
                Valid := TRUE;
                Error                   := _AxisReference^.Telegram111_In.ZSW1.faultPresent;
                ErrorID                 := TO_WORD(_AxisReference^.Telegram111_In.Fault_Code);
                ErrorStop               := DriveState = AXOpen.Components.Drives.eAxoDriveState#ErrorStop;;
                Disabled                := DriveState = AXOpen.Components.Drives.eAxoDriveState#Disabled;
                Stopping                := DriveState = AXOpen.Components.Drives.eAxoDriveState#Stopping;
                Homing                  := DriveState = AXOpen.Components.Drives.eAxoDriveState#Homing;
                Standstill              := DriveState = AXOpen.Components.Drives.eAxoDriveState#Standstill;
                DiscreteMotion          := DriveState = AXOpen.Components.Drives.eAxoDriveState#DiscreteMotion;
                ContinuousMotion        := DriveState = AXOpen.Components.Drives.eAxoDriveState#ContinuousMotion;
                SynchronizedMotion      := DriveState = AXOpen.Components.Drives.eAxoDriveState#SynchronizedMotion;
            END_IF;
        END_METHOD

        ///<summary>
        /// This method returns in detail the status of the axis with respect to the motion currently in progress.
        ///<summary>
        VAR INTERNAL
            MC_ReadMotionStateEnable_PV        : 	BOOL := FALSE;		//Enable - previous value
            MC_ReadMotionStateErrorID          : 	WORD;
            MC_ReadMotionStateCycle			: 	ULINT;
            MC_ReadMotionStateValue			: 	LINT;
            MC_ReadMotionStateValid			: 	BOOL;
        END_VAR
        METHOD PUBLIC OVERRIDE MC_ReadMotionState
            VAR_INPUT
                AxisRef         :   AXOpen.Components.Abstractions.Drives.IAxoAxisReference;
                Enable          :   BOOL;                       //  Get the value of the parameter continuously while enabled
                Source          :   AXOpen.Components.Abstractions.Drives.eAxoSource;                 //  Defines the source of the relevant data: CommandedValue;SetValue, ActualValue.
            END_VAR
            VAR_OUTPUT
                Valid           :   BOOL;                       //  A valid output is available at the method
                Busy            :   BOOL;                       //  The method is not finished and new output values are to be expected
                Error           :   BOOL;                       //  Signals that an error has occurred within the method
                ErrorID         :   WORD;                       //  Error identification
                ConstantVelocity:   BOOL;                       //  Velocity is constant. Velocity may be 0. For the actual value a window is applicable (window is vendor specific)
                Accelerating    :   BOOL;                       //  Increasing the absolute value of the velocity
                Decelerating    :   BOOL;                       //  Decreasing the absolute value of the velocity
                DirectionPositive:  BOOL;                       //  Signals that the position is increasing
                DirectionNegative:  BOOL;                       //  Signals that the position is decreasing
            END_VAR
            VAR
                _AxisReference :  REF_TO AXOpen.Components.Festo.Drives.AxoCmmtAsAxisReference;
                Dummy : BOOL;
            END_VAR

            _AxisReference ?= AxisRef;

            Messenger.ActivateOnCondition(ULINT#733,_AxisReference = NULL, eAxoMessageCategory#ProgrammingError);

            IF(_AxisReference = NULL) THEN
                RETURN;
            END_IF;
            IF Enable THEN
                Valid := TRUE;
                Error                   := _AxisReference^.Telegram111_In.ZSW1.faultPresent;
                ErrorID                 := TO_WORD(_AxisReference^.Telegram111_In.Fault_Code);
                ConstantVelocity        := FALSE;
                Accelerating            := _AxisReference^.Telegram111_In.ZSW1.axisAccelerates;
                Decelerating            := _AxisReference^.Telegram111_In.ZSW1.axisDecelerates;
                DirectionPositive       := _AxisReference^.Telegram111_In.POS_ZSW2.%X4;
                DirectionNegative       := _AxisReference^.Telegram111_In.POS_ZSW2.%X5;
             END_IF;
        END_METHOD

        ///<summary>
        /// This method reads information concerning an axis, like modes, inputs directly related to the axis,
        /// and certain status information.
        ///<summary>
        METHOD PUBLIC OVERRIDE MC_ReadAxisInfo
            VAR_INPUT
                AxisRef             :   AXOpen.Components.Abstractions.Drives.IAxoAxisReference;
                Enable              :   BOOL;                       //  Get the value of the parameter continuously while enabled
            END_VAR
            VAR_OUTPUT
                Valid               :   BOOL;                       //  A valid output is available at the method
                Busy                :   BOOL;                       //  The method is not finished and new output values are to be expected
                Error               :   BOOL;                       //  Signals that an error has occurred within the method
                ErrorID             :   WORD;                       //  Error identification
                HomeAbsSwitch       :   BOOL;                       //  Digital home switch input is active
                LimitSwitchPos      :   BOOL;                       //  Positive hardware end switch is active
                LimitSwitchNeg      :   BOOL;                       //  Negative hardware end switch is active
                Simulation          :   BOOL;                       //  Axis is in simulation mode (e.g. motor is simulated)
                CommunicationReady  :   BOOL;                         //  “Network” is initialized and ready for communication
                ReadyForPowerOn     :   BOOL;                       //  Drive is ready to be enabled (power on)
                PowerOn             :   BOOL;                       //  If TRUE shows that the power stage is switched ON
                IsHomed             :   BOOL;                       //  The absolute reference position is known for the axis (axis is homed)
                AxisWarning         :   BOOL;                       //  Warning(s) on the axis is present
            END_VAR
            VAR
                _AxisReference :  REF_TO AXOpen.Components.Festo.Drives.AxoCmmtAsAxisReference;
                Dummy : BOOL;
            END_VAR

            _AxisReference ?= AxisRef;

            Messenger.ActivateOnCondition(ULINT#734,_AxisReference = NULL, eAxoMessageCategory#ProgrammingError);

            IF(_AxisReference = NULL) THEN
                RETURN;
            END_IF;

            IF Enable THEN
                Valid := TRUE;
                Error                   := _AxisReference^.Telegram111_In.ZSW1.faultPresent;
                ErrorID                 := TO_WORD(_AxisReference^.Telegram111_In.Fault_Code);
                HomeAbsSwitch           := FALSE;
                LimitSwitchPos          := _AxisReference^.Telegram111_In.POS_ZSW1.%X9;
                LimitSwitchNeg          := _AxisReference^.Telegram111_In.POS_ZSW1.%X8;
                Simulation              := FALSE;
                CommunicationReady      := FALSE;
                ReadyForPowerOn         := _AxisReference^.Telegram111_In.ZSW1.readyForSwitchOn;
                PowerOn                 := _AxisReference^.Telegram111_In.ZSW1.operationEnabled;
                IsHomed                 := _AxisReference^.Telegram111_In.ZSW1.homePosSet;
                AxisWarning             := _AxisReference^.Telegram111_In.ZSW1.warningActive;
            END_IF;
        END_METHOD

        ///<summary>
        /// This method presents general axis errors not relating to the methods.
        /// (for instance axis errors, drive errors, communication errors)
        ///<summary>
        VAR INTERNAL
            MC_ReadAxisErrorEnable_PV        : 	BOOL := FALSE;		//Enable - previous value
            MC_ReadAxisErrorErrorID          : 	WORD;
            MC_ReadAxisErrorCycle			: 	ULINT;
            MC_ReadAxisErrorValue			: 	LINT;
            MC_ReadAxisErrorValid			: 	BOOL;
            LastMessageCode :   ULINT;
        END_VAR
        METHOD PUBLIC OVERRIDE MC_ReadAxisError
            VAR_INPUT
                AxisRef         :   AXOpen.Components.Abstractions.Drives.IAxoAxisReference;
                Enable          :   BOOL;                       //  Get the value of the parameter continuously while enabled
            END_VAR
            VAR_OUTPUT
                Valid           :   BOOL;                       //  A valid output is available at the method
                Busy            :   BOOL;                       //  The method is not finished and new output values are to be expected
                Error           :   BOOL;                       //  Signals that an error has occurred within the method
                ErrorID         :   WORD;                       //  Error identification
                AxisErrorID     :   DWORD;                      //  The value of the axis error. These values are vendor specific
            END_VAR
            VAR
                _AxisReference :  REF_TO AXOpen.Components.Festo.Drives.AxoCmmtAsAxisReference;
                Dummy : BOOL;
                _category  :   AXOpen.Messaging.eAxoMessageCategory;
            END_VAR

            _AxisReference ?= AxisRef;

            Messenger.ActivateOnCondition(ULINT#735,_AxisReference = NULL, eAxoMessageCategory#ProgrammingError);

            IF(_AxisReference = NULL) THEN
                RETURN;
            END_IF;

            IF Enable AND NOT MC_ReadAxisErrorEnable_PV AND State = UINT#0 THEN
                _AxisReference^.Status.CurrentMotionTaskId := AXOpen.Components.Drives.eAxoMotionTaskId#Axo_ReadAxisError;
                _AxisReference^.Data.Cycle := _AxisReference^.Data.Cycle + ULINT#2;
                MC_ReadAxisErrorCycle := _AxisReference^.Data.Cycle ;
            END_IF;

            IF Enable THEN
                IF State = UINT#0 THEN
                    Busy := TRUE;
                    MC_ReadAxisErrorErrorID := WORD#16#0000;
                    Parametrization.Inputs.Enable := FALSE;
                    State := UINT#310;
                END_IF;
                IF State = UINT#310 THEN
                    Busy := TRUE;
                    Parametrization.Inputs.Enable := TRUE;
                    Parametrization.Inputs.ReadWrite   := FALSE;
                    Parametrization.Inputs.ParameterNo := 12306;
                    Parametrization.Inputs.Subindex    := 0;
                    Parametrization.Inputs.AxisNo  := BYTE#1;
                    Parametrization.Inputs.HardwareId  := _AxisReference^.Data.MAP_HW_ID;
                    IF Parametrization.Outputs.Done AND NOT Parametrization.Outputs.Error THEN
                        MC_ReadAxisErrorValid := TRUE;
                        MC_ReadAxisErrorValue := Parametrization.Outputs.ValueReadLINT;
                        State := UINT#311;
                    END_IF;
                    IF Parametrization.Outputs.Error THEN
                        MC_MoveVelocityErrorID := WORD#813;
                        State := UINT#319;
                    END_IF;
                END_IF;
                IF State = UINT#311 THEN
                    Busy := TRUE;
                    Parametrization.Inputs.Enable := FALSE;
                    Parametrization.Inputs.ReadWrite   := FALSE;
                    IF  NOT Parametrization.Outputs.Done THEN
                        State := UINT#310;
                    END_IF;
                END_IF;
                IF State = UINT#319 THEN
                    Error := TRUE;
                END_IF;

                IF State>=UINT#310 AND State<UINT#317 THEN
                    IF _AxisReference^.Data.Cycle <> MC_ReadAxisErrorCycle THEN
                        _AxisReference^.Data.Cycle := _AxisReference^.Data.Cycle - ULINT#1;
                        State := UINT#319;
                    END_IF;
                END_IF;
            END_IF;

            IF NOT Enable AND MC_ReadAxisErrorEnable_PV  THEN
                _AxisReference^.Status.CurrentMotionTaskId := AXOpen.Components.Drives.eAxoMotionTaskId#Axo_None;
                MC_ReadAxisErrorErrorID := WORD#0;
                MC_ReadAxisErrorCycle := ULINT#0;
                MC_ReadAxisErrorValid := FALSE;
                MC_ReadAxisErrorValue := LINT#0;
                State := UINT#0;
            END_IF;

            ErrorID := MC_ReadAxisErrorErrorID;
            Valid := MC_ReadAxisErrorValid;
            MC_ReadAxisErrorEnable_PV := Enable;

            Messenger.ActivateOnCondition(LastMessageCode,Enable AND Valid AND LastMessageCode = TO_ULINT(MC_ReadAxisErrorValue), eAxoMessageCategory#Error);
            IF NOT Messenger.IsActive THEN
                LastMessageCode := TO_ULINT(MC_ReadAxisErrorValue);
            END_IF;
        END_METHOD

        ///<summary>
        /// This method makes the transition from the state ‘ErrorStop’ to ‘Standstill’ or ‘Disabled’ by resetting all
        /// internal axis-related errors – it does not affect the output of the other methods.
        ///<summary>
        VAR INTERNAL
            MC_ResetExecute_PV					: 	BOOL := FALSE;		//Execute - previous value
            MC_ResetPower_PV					: 	BOOL := FALSE;		//Execute - previous value
        END_VAR
        METHOD PUBLIC OVERRIDE MC_Reset
            VAR_INPUT
                AxisRef         :   AXOpen.Components.Abstractions.Drives.IAxoAxisReference;
                Execute         :   BOOL;                       //  Resets all internal axis-related error
            END_VAR
            VAR_OUTPUT
                Done            :   BOOL;                       //  ‘Standstill’ or ‘Disabled’ state is reached
                Busy            :   BOOL;                       //  The method is not finished and new output values are to be expected
                Error           :   BOOL;                       //  Signals that an error has occurred within the method
                ErrorID         :   WORD;                       //  Error identification
            END_VAR
            VAR
                _AxisReference :  REF_TO AXOpen.Components.Festo.Drives.AxoCmmtAsAxisReference;
                Dummy : BOOL;
            END_VAR

            _AxisReference ?= AxisRef;

            Messenger.ActivateOnCondition(ULINT#736,_AxisReference = NULL, eAxoMessageCategory#ProgrammingError);

            IF(_AxisReference = NULL) THEN
                RETURN;
            END_IF;

            IF Execute AND NOT MC_ResetExecute_PV THEN
                _AxisReference^.Telegram111_Out.STW1.StartHoming := FALSE;
                _AxisReference^.Telegram111_Out.POS_STW1.MDI_MOD := FALSE;
                _AxisReference^.Telegram111_Out.POS_STW1.PosModulo := FALSE;
                _AxisReference^.Telegram111_Out.POS_STW1.NegModulo := FALSE;
                _AxisReference^.Telegram111_Out.POS_STW1.SetupMode := FALSE;
                _AxisReference^.Telegram111_Out.POS_STW1.MDI_Activate := FALSE;
                _AxisReference^.Telegram111_Out.POS_STW2.Trackingmode := FALSE;
                _AxisReference^.Telegram111_Out.POS_STW2.jog_inc := FALSE;
                _AxisReference^.Telegram111_Out.POS_STW1.travBlockBit0 := FALSE;
                _AxisReference^.Telegram111_Out.POS_STW1.travBlockBit1 := FALSE;
                _AxisReference^.Telegram111_Out.POS_STW1.travBlockBit2 := FALSE;
                _AxisReference^.Telegram111_Out.POS_STW1.travBlockBit3 := FALSE;
                _AxisReference^.Telegram111_Out.POS_STW1.travBlockBit4 := FALSE;
                _AxisReference^.Telegram111_Out.POS_STW1.travBlockBit5 := FALSE;
                _AxisReference^.Telegram111_Out.POS_STW1.travBlockBit6 := FALSE;
                _AxisReference^.Telegram111_Out.STW2.TravelToFixStop := FALSE;
                Parametrization.Inputs.Enable := FALSE;
                State := UINT#320;
            END_IF;

            IF Execute THEN
                IF State = UINT#320 THEN
                    Busy := TRUE;
                    THIS.Restore();
                    THIS.AxoReset_Task.Invoke();
                    State := UINT#321;
                END_IF;
                IF State = UINT#321 THEN
                    Busy := TRUE;
                    MC_ResetPower_PV := AxoPower_Task.IsSwitchedOn();
                    State := UINT#322;
                END_IF;
                IF State = UINT#322 THEN
                    Busy := TRUE;
                    THIS.AxoPower_Task.SwitchOff();
                    IF THIS.AxoPower_Task.IsSwitchedOff() THEN
                        State := UINT#323;
                    END_IF;
                END_IF;
                IF State = UINT#323 THEN
                    Busy := TRUE;
                    _AxisReference^.Telegram111_Out.STW1.acknowledgeFault := TRUE;
                    State := UINT#324;
                END_IF;
                IF State = UINT#324 THEN
                    Busy := TRUE;
                    IF  NOT _AxisReference^.Telegram111_In.ZSW1.faultPresent THEN
                        State := UINT#325;
                    END_IF;
                    IF  _AxisReference^.Telegram111_In.ZSW1.faultPresent  AND THIS.AxoReset_Task.Duration >=T#2S THEN
                        State := UINT#329;
                    END_IF;
                END_IF;
                IF State = UINT#325 THEN
                    Busy := TRUE;
                    IF MC_ResetPower_PV THEN
                        State := UINT#326;
                    ELSE
                        State := UINT#327;
                    END_IF;
                END_IF;
                IF State = UINT#326 THEN
                    Busy := TRUE;
                    THIS.AxoPower_Task.SwitchOn();
                    IF THIS.AxoPower_Task.IsSwitchedOn() THEN
                        State := UINT#327;
                    END_IF;
                END_IF;
                IF State = UINT#327 THEN
                    _AxisReference^.Telegram111_Out.STW1.acknowledgeFault := FALSE;
                    Done := TRUE;
                END_IF;
                IF State = UINT#329 THEN
                    _AxisReference^.Telegram111_Out.STW1.acknowledgeFault := FALSE;
                    Error := TRUE;
                    ErrorID := TO_WORD(_AxisReference^.Telegram111_In.Fault_Code);
                END_IF;
            END_IF;

            IF NOT Execute AND MC_ResetExecute_PV THEN
                State := UINT#0;
            END_IF;

            MC_ResetExecute_PV := Execute;
        END_METHOD

        METHOD PUBLIC OVERRIDE Restore
            MC_HomeExecute_PV					:= FALSE;
            MC_HomeErrorID					    := WORD#0;
            MC_HomeCycle					    := ULINT#0;
            MC_StopExecute_PV					:= FALSE;
            MC_StopErrorID					    := WORD#0;
            MC_StopCycle					    := ULINT#0;
            MC_HaltExecute_PV					:= FALSE;
            MC_HaltErrorID					    := WORD#0;
            MC_HaltCycle					    := ULINT#0;
            MC_MoveAbsoluteExecute_PV			:= FALSE;
            MC_MoveAbsoluteErrorID				:= WORD#0;
            MC_MoveAbsoluteCycle				:= ULINT#0;
            MC_MoveAbsoluteContinuousUpdate_SV  := FALSE;
            MC_MoveAbsolutePosition_PV          := LREAL#0.0;
            MC_MoveAbsoluteVelocity_PV          := LREAL#0.0;
            MC_MoveAbsoluteAcceleration_PV      := LREAL#0.0;
            MC_MoveAbsoluteDeceleration_PV      := LREAL#0.0;
            MC_MoveAbsoluteJerk_PV              := LREAL#0.0;
            MC_MoveAbsoluteDirection_PV         := AXOpen.Components.Abstractions.Drives.eAxoDriveDirection#CurrentDirection;
            MC_MoveRelativeExecute_PV			:= FALSE;
            MC_MoveRelativeErrorID				:= WORD#0;
            MC_MoveRelativeCycle				:= ULINT#0;
            MC_MoveRelativeContinuousUpdate_SV  := FALSE;
            MC_MoveRelativeDistance_PV          := LREAL#0.0;
            MC_MoveRelativeVelocity_PV          := LREAL#0.0;
            MC_MoveRelativeAcceleration_PV      := LREAL#0.0;
            MC_MoveRelativeDeceleration_PV      := LREAL#0.0;
            MC_MoveRelativeJerk_PV              := LREAL#0.0;
            MC_MoveAdditiveExecute_PV			:= FALSE;
            MC_MoveAdditiveErrorID				:= WORD#0;
            MC_MoveAdditiveCycle				:= ULINT#0;
            MC_MoveAdditiveContinuousUpdate_SV  := FALSE;
            MC_MoveAdditiveDistance_PV          := LREAL#0.0;
            MC_MoveAdditiveVelocity_PV          := LREAL#0.0;
            MC_MoveAdditiveAcceleration_PV      := LREAL#0.0;
            MC_MoveAdditiveDeceleration_PV      := LREAL#0.0;
            MC_MoveAdditiveJerk_PV              := LREAL#0.0;
            MC_MoveVelocityExecute_PV			:= FALSE;
            MC_MoveVelocityErrorID				:= WORD#0;
            MC_MoveVelocityCycle				:= ULINT#0;
            MC_MoveVelocityContinuousUpdate_SV  := FALSE;
            MC_MoveVelocityVelocity_PV          := LREAL#0.0;
            MC_MoveVelocityAcceleration_PV      := LREAL#0.0;
            MC_MoveVelocityDeceleration_PV      := LREAL#0.0;
            MC_MoveVelocityJerk_PV              := LREAL#0.0;
            MC_MoveVelocityDirection_PV         := AXOpen.Components.Abstractions.Drives.eAxoDriveDirection#CurrentDirection;
            MC_TorqueControlExecute_PV			:= FALSE;
            MC_TorqueControlErrorID				:= WORD#0;
            MC_TorqueControlCycle				:= ULINT#0;
            MC_TorqueControlContinuousUpdate_SV := FALSE;
            MC_TorqueControlTorque_PV           := LREAL#0.0;
            MC_TorqueControlTorqueRamp_PV       := LREAL#0.0;
            MC_TorqueControlPositionLimit_PV    := LREAL#0.0;
            MC_TorqueControlVelocity_PV         := LREAL#0.0;
            MC_TorqueControlAcceleration_PV     := LREAL#0.0;
            MC_TorqueControlDeceleration_PV     := LREAL#0.0;
            MC_TorqueControlJerk_PV             := LREAL#0.0;
            MC_TorqueControlDirection_PV        := AXOpen.Components.Abstractions.Drives.eAxoDriveDirection#CurrentDirection;
            MC_SetPositionExecute_PV			:= FALSE;
            MC_SetPositionErrorID				:= WORD#0;
            MC_SetPositionCycle					:= ULINT#0;
            MC_SetPositionActualPosition        := LINT#0;
            MC_ReadParameterEnable_PV           := FALSE;
            MC_ReadParameterErrorID             := WORD#0;
            MC_ReadParameterCycle			    := ULINT#0;
            MC_ReadParameterValue			    := LINT#0;
            MC_ReadParameterValid			    := FALSE;
            MC_ReadRealParameterEnable_PV       := FALSE;
            MC_ReadRealParameterErrorID         := WORD#0;
            MC_ReadRealParameterCycle			:= ULINT#0;
            MC_ReadRealParameterValue			:= REAL#0.0;
            MC_ReadRealParameterValid			:= FALSE;
            MC_ReadBoolParameterEnable_PV       := FALSE;
            MC_ReadBoolParameterErrorID         := WORD#0;
            MC_ReadBoolParameterCycle			:= ULINT#0;
            MC_ReadBoolParameterValue			:= FALSE;
            MC_ReadBoolParameterValid			:= FALSE;
            MC_WriteParameterExecute_PV         := FALSE;
            MC_WriteParameterErrorID            := WORD#0;
            MC_WriteParameterCycle			    := ULINT#0;
            MC_WriteRealParameterExecute_PV     := FALSE;
            MC_WriteRealParameterErrorID        := WORD#0;
            MC_WriteRealParameterCycle			:= ULINT#0;
            MC_WriteBoolParameterExecute_PV     := FALSE;
            MC_WriteBoolParameterErrorID        := WORD#0;
            MC_WriteBoolParameterCycle			:= ULINT#0;
            MC_ReadDigitalInputEnable_PV        := FALSE;
            MC_ReadDigitalInputErrorID          := WORD#0;
            MC_ReadDigitalInputCycle			:= ULINT#0;
            MC_ReadDigitalInputValue			:= FALSE;
            MC_ReadDigitalInputValid			:= FALSE;
            MC_ReadDigitalOutputEnable_PV       := FALSE;
            MC_ReadDigitalOutputErrorID         := WORD#0;
            MC_ReadDigitalOutputCycle			:= ULINT#0;
            MC_ReadDigitalOutputValue			:= FALSE;
            MC_ReadDigitalOutputValid			:= FALSE;
            MC_WriteDigitalOutputExecute_PV     := FALSE;
            MC_WriteDigitalOutputErrorID        := WORD#0;
            MC_WriteDigitalOutputCycle			:= ULINT#0;
            MC_ReadStatusEnable_PV				:= FALSE;
            MC_ReadStatusDone_PV				:= FALSE;
            MC_ReadStatusStateNumber			:= INT#0;
            MC_ReadMotionStateEnable_PV         := FALSE;
            MC_ReadMotionStateErrorID           := WORD#0;
            MC_ReadMotionStateCycle			    := ULINT#0;
            MC_ReadMotionStateValue			    := LINT#0;
            MC_ReadMotionStateValid			    := FALSE;
            MC_ReadAxisErrorEnable_PV           := FALSE;
            MC_ReadAxisErrorErrorID             := WORD#0;
            MC_ReadAxisErrorCycle			    := ULINT#0;
            MC_ReadAxisErrorValue			    := LINT#0;
            MC_ReadAxisErrorValid			    := FALSE;
            LastMessageCode                     := ULINT#0;
            MC_ResetExecute_PV				    := FALSE;
            MC_ResetPower_PV				    := FALSE;

            _AxisRefExt.Data.Cycle              := ULINT#0;
            State                               := UINT#0;
            DriveStatus.Action.Id := UINT#0;
            DriveStatus.Error.Id  := UINT#0;
            Messenger.Restore();
            TaskMessenger.Restore();

            //AxoPower_Task.Restore();
            AxoStop_Task.Restore();
            AxoHalt_Task.Restore();
            AxoHome_Task.Restore();
            AxoMoveAbsolute_Task.Restore();
            AxoMoveRelative_Task.Restore();
            AxoMoveAdditive_Task.Restore();
            AxoMoveVelocity_Task.Restore();
            AxoTorqueControl_Task.Restore();
            AxoSetPosition_Task.Restore();
            AxoSetOverride_Task.SwitchOff();
            AxoReadParameter_Task.SwitchOff();
            AxoReadRealParameter_Task.SwitchOff();
            AxoReadBoolParameter_Task.SwitchOff();
            AxoWriteParameter_Task.Restore();
            AxoWriteRealParameter_Task.Restore();
            AxoWriteBoolParameter_Task.Restore();
            AxoReadDigitalInput_Task.SwitchOff();
            AxoReadDigitalOutput_Task.SwitchOff();
            AxoWriteDigitalOutput_Task.Restore();
            AxoReadActualPosition_Task.SwitchOff();
            AxoReadActualVelocity_Task.SwitchOff();
            AxoReadActualTorque_Task.SwitchOff();
            AxoReadStatus_Task.SwitchOff();
            AxoReadMotionState_Task.SwitchOff();
            AxoReadAxisInfo_Task.SwitchOff();
            AxoReadAxisError_Task.SwitchOff();
            AxoReset_Task.Restore();
            AxoJogPositive.RemoteSwitchOn := FALSE;
            AxoJogPositive.StartMotion := FALSE;
            AxoJogPositive.StopMotion := FALSE;
            AxoJogNegative.RemoteSwitchOn := FALSE;
            AxoJogNegative.StartMotion := FALSE;
            AxoJogNegative.StopMotion := FALSE;

            RestoreTask.DoneWhen(TRUE);

            SUPER.Restore();
        END_METHOD
    END_CLASS
END_NAMESPACE

(* ---- AxoCmmtAsParameterIn.st ---- *)
NAMESPACE AXOpen.Components.Festo.Drives
    {S7.extern=ReadWrite}
    CLASS AxoCmmtAsParameterIn
        (******************* IndraDrive configuration  ***********************
        Master communication; Fieldbus settings:
        Parameter chanel 10Bytes / 5 Words I/O
        *)
        VAR PUBLIC
            Datalength	:	BYTE;	//Length of  transfer data*)
            FL_0		:	BOOL;	//Length userdata bit 0
            FL_1		:	BOOL;	//Length userdata bit 1
            FL_2		:	BOOL;	//Length userdata bit 2
            FL_3		:	BOOL;	//Length userdata bit 3
            ToggleBit	:	BOOL;	//Toggle bit
            LastBit		:	BOOL;	//Last bit
            Failure		:	BOOL;	//Failure while communication
            Reserve		:	BOOL;	//Reserve
            DataWord_0	:	WORD;	//Data WORD 0
            DataWord_1	:	WORD;	//Data word 1
            DataWord_2	:	WORD;	//Data word 2
            DataWord_3	:	WORD;	//Data word 3
        END_VAR
    END_CLASS
 END_NAMESPACE

(* ---- AxoCmmtAsParameterOut.st ---- *)
NAMESPACE AXOpen.Components.Festo.Drives
    {S7.extern=ReadWrite}
    CLASS AxoCmmtAsParameterOut
        (******************* IndraDrive configuration  ***********************
        Master communication; Fieldbus settings:
        Parameter chanel 10Bytes / 5 Words I/O
        *)
        VAR PUBLIC
            Datalength		:	BYTE := BYTE#04;//Length of transfer data
            FL_0			:	BOOL;			//Length userdata bit 0
            FL_1			:	BOOL;			//Length userdata bit 1
            FL_2			:	BOOL;			//Length userdata bit 2
            FL_3			:	BOOL;			//Length userdata bit 3
            ToggleBit		:	BOOL;			//Toggle bit
            LastBit			:	BOOL;			//Last bit
            Initalisation	:	BOOL := TRUE;	//Initialisation
            Reserve			:	BOOL;			//Reserve
            Index			:	WORD;			//Index number
            Subindex		:	BYTE;			//Subindex number
            Axis			:	BYTE;			//Axis number
            DataWord_0		:	WORD;			//Data word 0
            DataWord_1		:	WORD;			//Data word 1
        END_VAR
    END_CLASS
END_NAMESPACE
